FUNCTION_BLOCK FB_LamparaComputada_LD
VAR_INPUT
    ReiniciaContador: BOOL;
    ManiobrasTotales: UINT := 2;
    TiempoEncendido: REAL := 2.0;
END_VAR
VAR_OUTPUT
    LamparaHabilitada: BOOL;
    ManiobrasPendientes: UINT;
    TiempoPendiente: REAL;
END_VAR
VAR
    Lampara AT %Q*: BOOL;
    Pulsador AT %I*: BOOL;
    
    Contador: CTD := (CV := ManiobrasTotales);
    Temporizador: TON;

    Memoria: RS;
    Resultado: REAL;
    Tiempo: TIME;
END_VAR

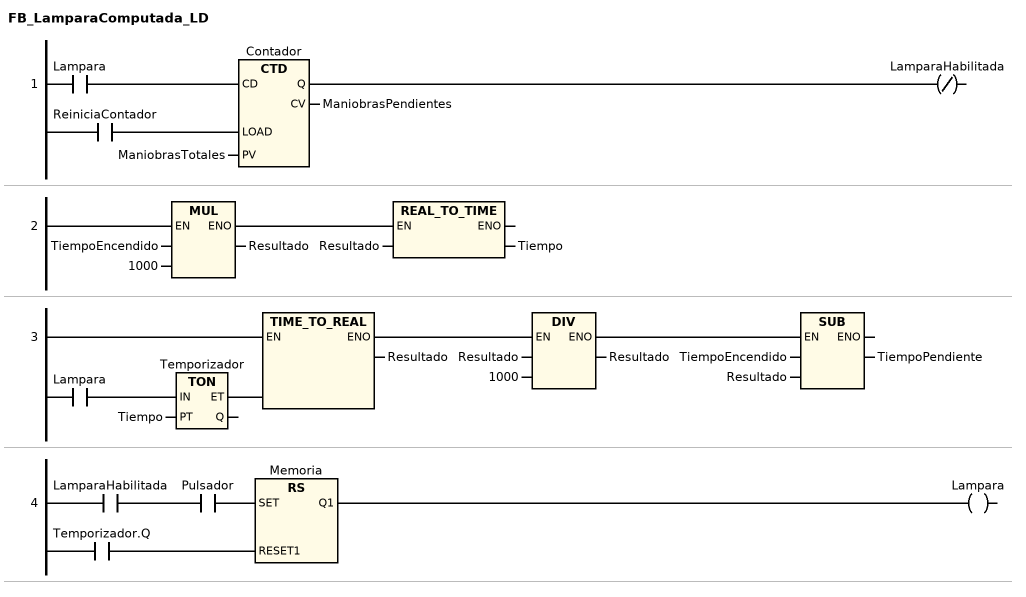
// NETWORK 1
Contador(CD := Lampara, LOAD := ReiniciaContador, PV := ManiobrasTotales, CV => ManiobrasPendientes); // CTD
LamparaHabilitada := NOT Contador.Q;

// NETWORK 2
Resultado := TiempoEncendido * 1000;
Tiempo := REAL_TO_TIME(Resultado);

// NETWORK 3
Temporizador(IN := Lampara, PT := Tiempo); // TON
Resultado := TIME_TO_REAL(Temporizador.ET);
Resultado := Resultado / 1000;
TiempoPendiente := TiempoEncendido - Resultado;

// NETWORK 4
Memoria(SET := LamparaHabilitada AND Pulsador, RESET1 := Temporizador.Q); // RS
Lampara := Memoria.Q1;

END_FUNCTION_BLOCK

(* stored: Version 1.1.0.1, ProductVersion 3.1.4024.15
   POU FB_LamparaComputada_LD: Id {41ef2a50-6ccd-433b-b47c-8214546b0362}, SpecialFunc None *)
